{attribute 'GeneratedUsingTerminal: EQ3204-0002-0021'}
{attribute addProperty BoxType "EQ3204-0002-0021"}
{attribute addProperty Id "StatusAT %I*Status_F2CE6D917ValueAT %I*INT2"}
{attribute addProperty CRC "1245267073"}
{attribute addProperty Size "9"}
TYPE RTD_RTDInputs_Channel_4A394481 :
STRUCT
	{attribute addProperty Name "Status"}
	Status AT %I* : Status_F2CE6D91;
	{attribute addProperty Name "Value"}
	Value AT %I* : INT;
END_STRUCT
END_TYPE

(* stored: Version 1.2.0.0, ProductVersion 3.1.4024.9
   DUT RTD_RTDInputs_Channel_4A394481: Id {350c98ff-d87a-4280-bd49-8e031ff5f5ef} *)
